PROGRAM MAIN
VAR
	counter:INT:=0;
END_VAR

counter:=counter+1;

MAIN_1();
MAIN_2();

END_PROGRAM

(* stored: Version 1.1.0.1, ProductVersion 3.1.4024.9
   POU MAIN: Id {f1e8bf76-a09f-4110-812f-d2f89db87cce}, SpecialFunc None *)
